FUNCTION_BLOCK WAGOConvBeltModel (* Model a conveyor *)
  (* Standard: 61499-2 *)
  (* Version 0.2, 2003-12-04, JHC, Rockwell Automation, Renamed for better indexing. *)
  (* Compiler header: package fb.rt.wago; #include <stdio.h> *)
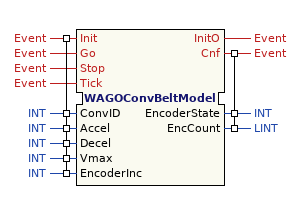
  EVENT_INPUT
    Init WITH ConvID, Vmax, Accel, Decel, EncoderInc; (* Initialization Request *)
    Go;
    Stop;
    Tick;
  END_EVENT
  EVENT_OUTPUT
    InitO; (* Initialization Confirm *)
    Cnf WITH EncoderState, EncCount; (* Execution Confirmation *)
  END_EVENT
  VAR_INPUT
    ConvID : INT; (* Conveyor ID *)
    Accel : INT; (* Acceleration of conveyor speed *)
    Decel : INT; (* Decceleration of conveyor speed *)
    Vmax : INT; (* Maximum velocity *)
    EncoderInc : INT; (* Length of conveyor travelled for each encoder transition (mm) *)
  END_VAR
  VAR_OUTPUT
    EncoderState : INT := 0;
    EncCount : LINT := 0; (* Used internally for plant stuff *)
  END_VAR
  VAR
    V : INT; (* velocity (mm per sec) of conveyor belt *)
    a : INT; (* current acceleration *)
    count : LINT; (* EncCount of conveyor (incremented every 50 mm) *)
    LastStateChangeCount : LINT; (* EncCount of last EncoderState Change *)
    stop : BOOL; (* Set if conveyor has come to a complete stop *)
  END_VAR
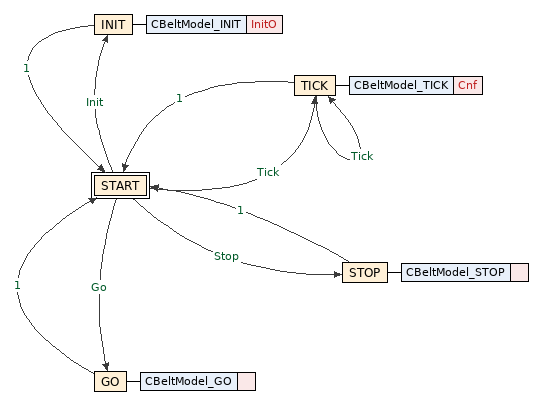
  EC_STATES
    START; (* Initial State *)
    INIT : CBeltModel_INIT -> InitO; (* Initialization *)
    GO : CBeltModel_GO;
    STOP : CBeltModel_STOP;
    TICK : CBeltModel_TICK -> Cnf;
  END_STATES
  EC_TRANSITIONS
    START TO INIT := Init;
    INIT TO START := 1;
    TICK TO START := 1;
    START TO STOP := Stop;
    START TO GO := Go;
    GO TO START := 1;
    STOP TO START := 1;
    START TO TICK := Tick;
    TICK TO TICK := Tick;
  END_TRANSITIONS
  ALGORITHM CBeltModel_INIT IN C: (* Initialization algorithm *)
 printf("CBeltModel_INIT: %d ConvID, %d Accel, %d Decel, %d Vmax, %d V, %lld count, %d stop\n", me->ConvID, me->Accel, me->Decel, me->Vmax, me->V, me->count, me->stop);
 me->V = 0 ;
 me->count = 0 ;
 me->stop = true ;
  END_ALGORITHM
  ALGORITHM CBeltModel_GO IN C: (* To start conveyor and to change conveyor's acceleration *)
 me->a = me->Accel ;
 me->stop = false ;
 printf("CBeltModel_GO[%d]: Conveyor Started (%d acc, %d dec, %d a, %c stop)\n",me->ConvID, me->Accel, me->Decel,me->a,me->stop);
  END_ALGORITHM
  ALGORITHM CBeltModel_STOP IN C: (* To stop the conveyor *)
 printf("CBeltModel_STOP[%d]: Conveyor Stopped.\n", me->ConvID);
 me->a = me->Decel;
  END_ALGORITHM
  ALGORITHM CBeltModel_TICK IN C: (* Called every 500msec *)
 if (me->V < me->Vmax && me->a >= 0)
 {
  //printf("Increasing speed (%d / %d = %d) + %d!!!\n", *a, 2, (*a+2),*V);
  me->V = me->V + (me->a / 2) ;
  //printf("CBeltModel_TICK[%d]: New speed: %d\n",*ID,*V);
  // to check value of V after the adjustment
  if (me->V > me->Vmax)
   me->V = me->Vmax ;
  else if( me->V < 0 )
   me->V = 0.0;
 }
 else if( me->a < 0 )
 {
  if (me->V > 0)
   me->V = me->V + (me->a / 2) ;
  else {
   me->stop = true ;
    me->a = 0 ;
   }
 }
 me->count = me->count + me->V ;
 //if( *ID == 0 )
 //printf("[CBM] (%lld / 50) >  %lld\n", me->count,  me->LastStateChangeCount);
 if( me->V >= 50 || (me->count / 50) >  me->LastStateChangeCount )
 {
  if( me->EncoderState != 0 ) me->EncoderState = 0;
  else me->EncoderState = 1;
  me->LastStateChangeCount = (me->count / 50);
  //printf("New Enccount = %lld\n",me->count);
 }
 me->EncCount = me->count ;  //updating EncCount
  END_ALGORITHM
END_FUNCTION_BLOCK
